TEXTLIST TextList
  0 = '0'
  1 = '1'
  2 = '3'
  4 = '5'
  6 = '6'
  7 = '7'
  8 = '8'
  9 = '9'
  10 = '10'
   = ''
END_TEXTLIST

(* stored: Version 1.1.0.1, ProductVersion 3.1.4024.15
   TextList TextList: Id {778c16fa-dae5-45ec-88b2-761b46dc7eee} *)
